# EPICS substitutions: db/Beckhoff_5XXX/ecmcEL5112_ABC.substitutions
file "ecmcEL5131-chX.template"
{
    pattern {CH_ID}
            {01   }
}
